(* PLC project Sin nombre, Desconocido Sin nombre 1 *)
(* stored: creationDateTime 2024-11-27T11:47:02, modificationDateTime 2024-11-27T12:10:59 *)

PROGRAM reles
  VAR
    Start : BOOL := fasle;
    Stop : BOOL := true;
    K1 : LOGLEVEL;
  END_VAR

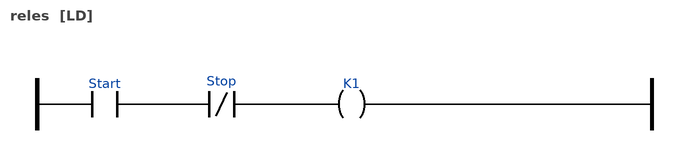
(* LD diagram, written out as Structured Text *)
K1 := Start AND NOT Stop;
END_PROGRAM

CONFIGURATION Config0
  RESOURCE Res0 ON PLC
    TASK task0(INTERVAL := T#20ms, PRIORITY := 0);
    PROGRAM instance0 WITH task0 : reles;
  END_RESOURCE
END_CONFIGURATION
